FUNCTION_BLOCK FB_ExtrusionSystemRev
VAR_INPUT
	bEnable 			: BOOL;
	bReset 				: BOOL;
	bExecuteExtrude		: BOOL;
	lrMMtoExtrude  		: LREAL;
	lrRetractionLength	: LREAL;
	lrFeedrate   		: LREAL;
	lrHotEndTempSP		: LREAL;
	lrHotEndTemp 		: LREAL;	
END_VAR
VAR_OUTPUT
	sStateDesc			: STRING;
	bExtrudeDone 	    : BOOL;
	bError				: BOOL;
	bExtruderReady		: BOOL;
	bExtruderMoving		: BOOL;
	iHotEndPowerLevel 	: INT;
	bFan				: BOOL;
	bEnableHotend		: BOOL;
	eErrorId			: UDINT;
END_VAR
VAR_IN_OUT
	ExtruderAxisRef			: AXIS_REF;
END_VAR
VAR
	nState					: UDINT := 0;
	nErrorState				: UDINT;
		
	RTrig_Reset				: R_TRIG;
	MC_Power_Extruder		: MC_Power;
	MC_Reset_Extruder 		: MC_Reset;
	MC_ZeroPos_Extruder		: MC_SetPosition;
	MC_Stop_Extruder 		: MC_Stop;
	MC_Move_Rel_Extruder 	: MC_MoveRelative;
	fbHotendTempController 	: FB_TempControl;
	
	bHeating				: BOOL := FALSE;
	bAtTempSP				: BOOL := FALSE;
	bMoveRelative			: BOOL := FALSE;
	fbSetPos				: MC_SetPosition;
	lrExtrudeDist  			: LREAL;
END_VAR

ExtruderAxisRef.ReadStatus();
RTrig_Reset(CLK:=bReset , Q=> );

MC_Power_Extruder(
	Axis:= ExtruderAxisRef, 
	Enable:= bExtruderReady, 
	Enable_Positive:= bExtruderReady, 
	Enable_Negative:= bExtruderReady, 
	Override:= , 
	BufferMode:= , 
	Options:= , 
	Status=> , 
	Busy=> , 
	Active=> , 
	Error=> bError, 
	ErrorID=> eErrorId);
	
fbHotendTempController(
		bEnableHeater:= bEnableHotEnd, 
		lrPV:= lrHotendTemp, 
		lrSP:= lrHotEndTempSP, 
		iOutput=> iHotEndPowerLevel, 
		bError=>bError, 
		eErrorId=> eErrorId,
		bEnableHotend=> bEnableHotend);
		
MC_Move_Rel_Extruder(
	Axis:= ExtruderAxisRef, 
	Execute:= bMoveRelative, 
	Distance:= lrExtrudeDist, 
	Velocity:= lrFeedrate, 
	Acceleration:= , 
	Deceleration:= , 
	Jerk:= , 
	BufferMode:= , 
	Options:= , 
	Done=> bExtrudeDone, 
	Busy=> , 
	Active=> bExtruderMoving , 
	CommandAborted=> , 
	Error=> bError, 
	ErrorID=> eErrorId);
	
//IF NOT bEnable THEN
//	nState := 10;
//END_IF

IF RTrig_Reset.CLK THEN
	nState := 100;
END_IF

IF lrHotendTemp >= (lrHotEndTempSP*0.98) THEN
	bAtTempSP := TRUE;
ELSE
	bAtTempSP := FALSE;
END_IF

	
CASE nState OF
	0:	// init
		sStateDesc := 'FB INIT';
		bExtrudeDone := FALSE;
		bError := FALSE;
		bExtruderMoving := FALSE;
		//GVL_AxisCtrl.bExtruder_AxisAbsMove := FALSE;
		iHotEndPowerLevel := 0;
		bFan := FALSE;
		nState := 10;
		
	10: // idle
		sStateDesc := 'IDLE';
		iHotEndPowerLevel := 0;
		bEnableHotEnd := FALSE;
		bExtruderReady := FALSE;
		bFan := FALSE;
		IF bEnable THEN 
			nState := 20;
		END_IF		

	20: // Turn on heater
		IF NOT bEnable THEN
			nState := 10;
		END_IF
		
		sStateDesc := 'START HEATING';
		bFan := TRUE;			
		bEnableHotend := TRUE;
		nState := 30;
		
	30: // Heating
		IF NOT bEnable THEN
			nState := 10;
		END_IF
		sStateDesc := 'HEATING TO REACH OPERATING TEMP';
		IF bAtTempSP THEN
			nState := 40;
		ELSE
			bExtruderReady := FALSE;	
		END_IF
		
	40: // Ready to Extrude
		IF NOT bEnable THEN
			nState := 10;
		END_IF
		
		IF bAtTempSP THEN
			sStateDesc := 'WAITING FOR MOVE COMMAND';
			bExtruderReady := TRUE;
			IF bExecuteExtrude THEN;
				nState := 50;
			END_IF
		ELSE
			bExtruderReady := FALSE;
			nState := 30;
		END_IF
		
	50: // Move Relative
		IF NOT bEnable THEN
			nState := 10;
		END_IF
		sStateDesc := 'EXTRUDING';
		lrExtrudeDist := lrMMtoExtrude;
		bMoveRelative := TRUE;
		IF bExtrudeDone THEN (* Requested Distance Extruded *)
			bExtrudeDone 	:= FALSE;
			bMoveRelative 	:= FALSE;
			nState := 60;
		END_IF
	60: // Retract
		sStateDesc := 'RETRACTING';
		IF NOT bEnable THEN
			nState := 10;
		END_IF
		lrExtrudeDist := lrRetractionLength * -1; (* Retract *)
		bMoveRelative := TRUE;
		IF bExtrudeDone THEN (* Requested Retraction Done *)
			bExtrudeDone 	:= FALSE;
			bMoveRelative 	:= FALSE;
			nState := 40;
		END_IF
			
	100: // Reset
		sStateDesc := 'RESET EXTRUDER AXIS';
		MC_Reset_Extruder(Axis:=ExtruderAxisRef, Execute:=TRUE);
		IF MC_Reset_Extruder.Done THEN
			nState := 10;
		END_IF
	999: //Error	
		
	ELSE
	sStateDesc := 'INVALID STATE';
	nState := 0;
END_CASE

END_FUNCTION_BLOCK

(* stored: Version 1.1.0.1, ProductVersion 3.1.4024.2
   POU FB_ExtrusionSystemRev: Id {84e7df3e-7b62-404d-8a1c-2d9f0ad66415}, SpecialFunc None *)
